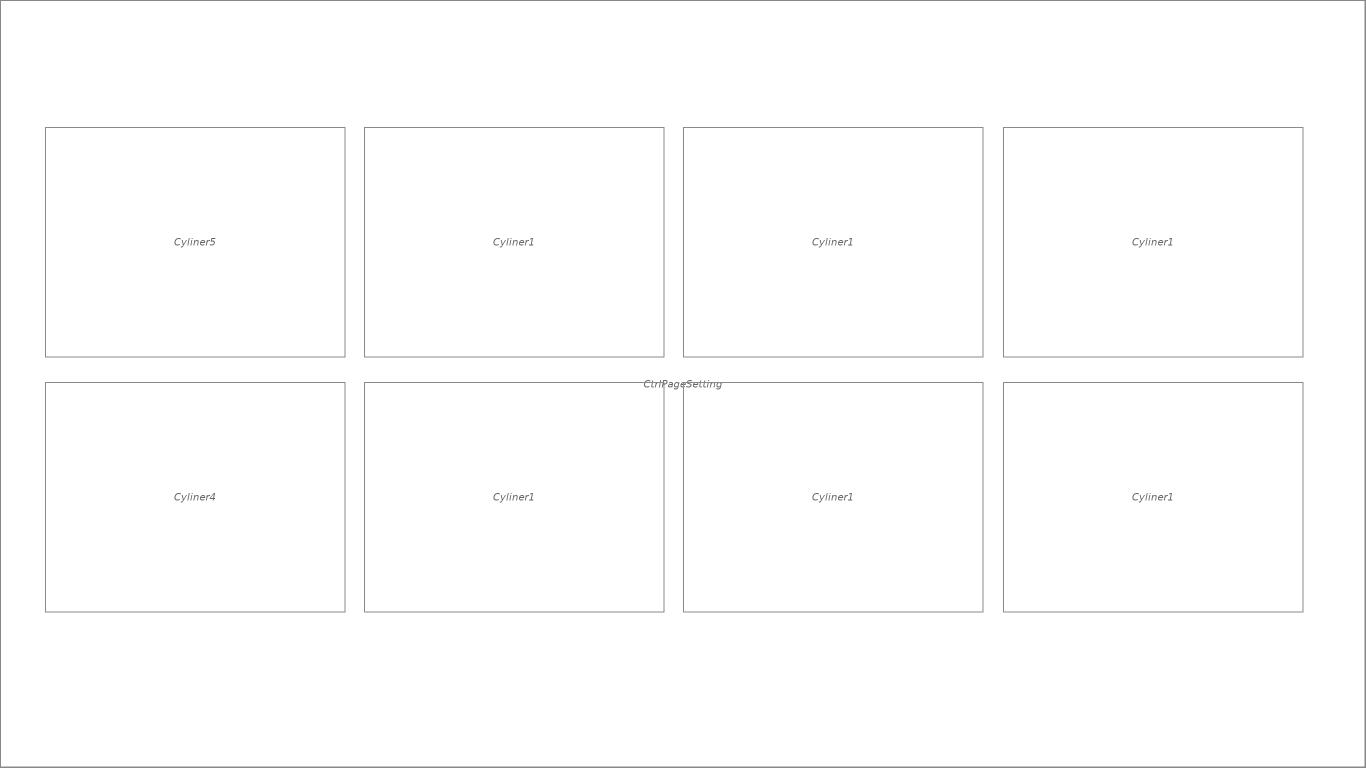
VISUALIZATION PageSetting_TakeUc  // 1366x768
    Frame (0,0 1366x768)
        shows CtrlPageSetting()
    Frame (364,127 300x230)
        shows Cyliner1(System := G_stSystem, Cylinder := G_arrCylinder[E_Cylinder.TakeUcPrevent], CylinderData := G_arrCylinderData[E_Cylinder.TakeUcPrevent])
    Frame (683,127 300x230)
        shows Cyliner1(System := G_stSystem, Cylinder := G_arrCylinder[E_Cylinder.TakeUcLift], CylinderData := G_arrCylinderData[E_Cylinder.TakeUcLift])
    Frame (1003,127 300x230)
        shows Cyliner1(System := G_stSystem, Cylinder := G_arrCylinder[E_Cylinder.TakeUcPush], CylinderData := G_arrCylinderData[E_Cylinder.TakeUcPush])
    Frame (45,382 300x230)
        shows Cyliner4(System := G_stSystem, Cylinder := G_arrCylinder[E_Cylinder.TakeUcRotate], CylinderData := G_arrCylinderData[E_Cylinder.TakeUcRotate])
    Frame (364,382 300x230)
        shows Cyliner1(System := G_stSystem, Cylinder := G_arrCylinder[E_Cylinder.TakeUcStandard], CylinderData := G_arrCylinderData[E_Cylinder.TakeUcStandard])
    Frame (683,382 300x230)
        shows Cyliner1(System := G_stSystem, Cylinder := G_arrCylinder[E_Cylinder.TakeUcElevator], CylinderData := G_arrCylinderData[E_Cylinder.TakeUcElevator])
    Frame (1003,382 300x230)
        shows Cyliner1(System := G_stSystem, Cylinder := G_arrCylinder[E_Cylinder.TakeUcPush1], CylinderData := G_arrCylinderData[E_Cylinder.TakeUcPush1])
    Frame (45,127 300x230)
        shows Cyliner5(System := G_stSystem, Cylinder := G_arrCylinder[E_Cylinder.TakeUcFrockClamp], CylinderData := G_arrCylinderData[E_Cylinder.TakeUcFrockClamp])
END_VISUALIZATION

(* stored: Version 1.1.0.1, ProductVersion 3.1.4024.3
   Visu PageSetting_TakeUc: Id {c056fc8c-53a5-4fec-8f19-de997e4f3d25} *)
